FUNCTION_BLOCK State2 EXTENDS AbstractState

METHOD Handle : BOOL
fbTON(IN := TRUE, PT := T#7s);
IF fbTON.Q THEN
	LogString(sString := 'Timer in State 2 fired. Changing State to State 1.');
	ipStatehandler.SetState(eNewState := E_STATES.eState1);
	fbTON(IN := FALSE);
END_IF
END_METHOD

END_FUNCTION_BLOCK

(* stored: Version 1.1.0.1, ProductVersion 3.1.4024.3
   POU State2: Id {e90cbb4f-15f1-4334-a8a3-9fa477e73284}, SpecialFunc None
   Method Handle: Id {5ace3522-1dad-456b-8124-c93d86626caf} *)
